// TwinCAT 3 PLC project lib
// Title: Test Framework
// Company: BA
// ProjectVersion: 1.0.0.0
// ProgramVersion: 3.1.4026.12
// libraries:
//   Tc2_Standard, * (Beckhoff Automation GmbH)
//   Tc2_System, * (Beckhoff Automation GmbH)
//   Tc2_Utilities, * (Beckhoff Automation GmbH)
//   Tc3_JsonXml, * (Beckhoff Automation GmbH)
// project tree:
//   FileIo/ FB_FileIO.TcPOU (not stored)
//   Project Information/ F_GetCompany.TcPOU, F_GetTitle.TcPOU (not stored), F_GetVersion.TcPOU
//   TestFramework/ FB_SimpleTest.TcPOU (not stored), FB_TestRunner.TcPOU, ITest.TcIO (not stored), TestResults.TcDUT (not stored)
//   Version/ Global_Version.TcGVL

// ---- Version/Global_Version.TcGVL
{attribute 'TcGenerated'}
{attribute 'no-analysis'}
{attribute 'linkalways'}
// This function has been automatically generated from the project information.
VAR_GLOBAL CONSTANT
	{attribute 'const_non_replaced'}
	stLibVersion_Test_Framework : ST_LibVersion := (iMajor := 1, iMinor := 0, iBuild := 0, iRevision := 0, nFlags := 0, sVersion := '1.0.0.0');
END_VAR

// ---- Project Information/F_GetCompany.TcPOU
// This function has been automatically generated from the project information.
{attribute 'signature_flag' := '1073741824'}
{attribute 'TcGenerated'}
{attribute 'no-analysis'}
FUNCTION F_GetCompany : WSTRING
VAR_INPUT
	
END_VAR

F_GetCompany := "BA";

END_FUNCTION

// ---- Project Information/F_GetVersion.TcPOU
// This function has been automatically generated from the project information.
{attribute 'signature_flag' := '1073741824'}
{attribute 'TcGenerated'}
{attribute 'no-analysis'}
FUNCTION F_GetVersion : ST_LibVersion
VAR_INPUT
	
END_VAR

F_GetVersion.iMajor := 1;
F_GetVersion.iMinor := 0;
F_GetVersion.iBuild := 0;
F_GetVersion.iRevision := 0;
F_GetVersion.sVersion := '1.0.0.0';
F_GetVersion.nFlags := 0;

END_FUNCTION

// ---- TestFramework/FB_TestRunner.TcPOU
FUNCTION_BLOCK FB_TestRunner
VAR_INPUT
END_VAR
VAR_OUTPUT
END_VAR
VAR
	i, nTestCount		: DINT;
	Tests				: ARRAY[0..9] OF ITest;
	sXmlString 			: STRING(1000);
	nState				: DINT;
	fbFileIo			: FB_FileIO;
END_VAR

METHOD AddTest : BOOL
VAR_INPUT
	Test		: ITest;
END_VAR
IF Test <> 0 THEN
	Tests[nTestCount] := Test;
	nTestCount := nTestCount + 1;
END_IF
END_METHOD

METHOD Execute : BOOL
VAR_INPUT
END_VAR
CASE nState OF
	0:
		IF i < nTestCount AND Tests[i] <> 0 THEN
			IF Tests[i].Execute() THEN
				i := i + 1;
			END_IF
		ELSE
			nState := 1;
		END_IF
	1:
		ToXml();
		nState := 2;
	2:
		// default write to root folder of the runtime (C:\ProgramData\Beckhoff\TwinCAT\3.1\Runtimes\UmRtTestFramework) 
		IF fbFileIo.WriteAllText('testresults.xml', sXmlString) THEN
			nState := 3;
		END_IF
	3:
		;
		
END_CASE

fbFileIo();
END_METHOD

METHOD ToXml : BOOL
VAR_INPUT
END_VAR
VAR
	fbXml 				: FB_XmlDomParser;
	objRoot 			: SXmlNode;
	objTestSuite 		: SXmlNode;
	objTestCase			: SXmlNode;
	objFailure			: SXmlNode;
	objFailureMsg		: SXmlNode;
	objAttribute 		: SXmlAttribute;
	
	j, nLength					: DINT;
	sCount, sTestName, sClass	: STRING;
	result						: TestResults;
END_VAR
objRoot := fbXml.GetDocumentNode();
objTestSuite := fbXml.AppendNode(objRoot, 'testsuite');
sCount := TO_STRING(nTestCount);
objAttribute := fbXml.AppendAttribute(objTestSuite, 'tests', sCount);

FOR j := 0 TO nTestCount - 1 DO
	sTestName := Tests[j].Name;
	sClass := Tests[j].ClassName;
	result := Tests[j].Result;
	objTestCase := fbXml.AppendNode(objTestSuite, 'testcase');
	objAttribute := fbXml.AppendAttribute(objTestCase, 'classname', sClass);
	objAttribute := fbXml.AppendAttribute(objTestCase, 'name', sTestName);
	IF NOT result.Passed THEN
		objFailure := fbXml.AppendChild(objTestCase, 'failure', result.Message, FALSE);
		objAttribute := fbXml.AppendAttribute(objFailure, 'type', 'assert');
	END_IF
END_FOR

nLength := fbXml.CopyDocument(sXmlString, SIZEOF(sXmlString));
END_METHOD

END_FUNCTION_BLOCK
